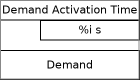
VISUALIZATION UI_Demand  // 140x80
VAR_IN_OUT
	hmi : Room_State_DemandHeating_Hmi;
END_VAR
    Rectangle (40,20 100x20), "%i s", text variable: hmi.nActivationTime
        OnMouseClick: write the text variable via Default
    Rectangle (0,0 140x20), "Demand Activation Time"
    Rectangle (0,50 140x30), "Demand", colour toggle: hmi.bDemandButton
        toggle hmi.bDemandButton
END_VISUALIZATION

(* stored: Version 1.1.0.1
   Visu UI_Demand: Id {c5fad084-02c2-40ed-a415-b87b6faec236} *)
